(*			
	RafalOS
	Rafał Osajda		12.11.2025		TC 4024.66
	Zbiór metod umożliwiające odczyt danych z hmi 
*)
INTERFACE ITF_HMIEMenu_HMI_Connector EXTENDS ITF_BaseControlElement_HMI_Connector

METHOD PUBLIC GetNumberOfActrivePreviewScreen : INT
VAR_INPUT
END_VAR
END_METHOD

METHOD PUBLIC GetNumberOfActriveScreen : INT
VAR_INPUT
END_VAR
END_METHOD

METHOD PUBLIC GetNumberOfAddedButton : INT
VAR_INPUT
END_VAR
END_METHOD

METHOD PUBLIC IsChangePage : BOOL
VAR_INPUT
END_VAR
END_METHOD

END_INTERFACE

(* stored: Version 1.1.0.1
   Itf ITF_HMIEMenu_HMI_Connector: Id {ad564c42-67d1-0387-1df7-423691c5bc76}
   Method GetNumberOfActrivePreviewScreen: Id {37bbb933-f165-04a3-37e4-a26af27797f3}
   Method GetNumberOfActriveScreen: Id {f18f1ac5-0cee-0dba-1fc3-ab4e5614410f}
   Method GetNumberOfAddedButton: Id {244a66b8-1190-0385-2576-d36189f23591}
   Method IsChangePage: Id {5977192d-eabb-02c2-2cc6-e8a135136555} *)
